{library public}

(* Common error values for communication blocks *)
TYPE COM_ERROR_VALUE :
(
	COM_ERR_NOT_ENABLED:=-1,						(* En signal is false or block is not enabled *)
	COM_ERR_NO_ERROR:=0,							(* No error *)

 	(* Level 1 Errors *)
	COM_ERR_LEVEL1,									(* The physical layer failed during communication *)
	COM_ERR_LEVEL1_TIME_OUT,						(* Time out in the physical layer *)

 	(* Level 2 Errors *)
	COM_ERR_NOT_ALLOCATED,							(* Instance not allocated *)
	COM_ERR_INSTANCE,								(* Instance address (station/device) number not set or wrong *)
	COM_ERR_LEVEL2_TIME_OUT,						(* Time out in communication with device *)
	COM_ERR_LEVEL2_ERROR,							(* Error during send/receive *)
	COM_ERR_CANCEL,									(* Current operation was cancelled *)

 	(* Level 3 Errors *)
	COM_ERR_TWO_INSTANCES_OF_COMMUNICATOR,			(* Two instances of the communicator block exist in the configuration remove one *)
	COM_ERR_CHECKSUM,								(* Checksum error during datagram transfer *)

	(* Level 5 Error *)
	COM_ERR_NO_VALID_FUNCTION						(* Calls to an unknown RPC function *)
);
END_TYPE
//  COM_ERR_NOT_ENABLED = '-1'

(* stored: Version 1.1.0.1, ProductVersion 3.1.4024.2
   EnumerationTextList COM_ERROR_VALUE: Id {e1bd82d2-ff44-4407-8d48-b3f359ffc33f} *)
